// TIA Portal V16 export
// export: Created 2022-07-21T09:35:14.5212503Z, ExportSetting WithDefaults, DisplayName Totally Integrated Automation Portal, DisplayVersion V16 Update 4, DisplayName TIA Portal Version Control Interface, DisplayVersion V16 Update 2, DisplayName TIA Portal Openness, DisplayVersion V16 Update 4, DisplayName SINAMICS Startdrive Advanced, DisplayVersion V16 Update 5, DisplayName SINAMICS Startdrive G130, G150, S120, S150, SINAMICS MV, S210, DisplayVersion V16 Update 5, DisplayName SINAMICS Startdrive G110M, G120, G120C, G120D, G120P, G115D, DisplayVersion V16 Update 5, DisplayName STEP 7 Professional, DisplayVersion V16 Update 4, DisplayName STEP 7 Safety, DisplayVersion V16, DisplayName WinCC Advanced, DisplayVersion V16 Update 4
FUNCTION_BLOCK "LAxisBasics_AxisBasics_SyncAxis"   // FB833, FBD
TITLE = SyncAxis / Obsługa SyncAxis
{ S7_Optimized_Access := 'TRUE' }
AUTHOR : ArSc
FAMILY : LAxisBasics
VERSION : 1.1
// stored: AutoNumber false, IsIECCheckEnabled false, IsRetainMemResEnabled false, MemoryReserve 100, SetENOAutomatically false, UDAEnableTagReadback false
   VAR_INPUT
      axis : TO_SynchronousAxis;
      powerEnable : Bool;
      powerStartMode : DInt := 1;
      powerStopMode : Int := 0;
      resetExecute : Bool;
      resetRestart : Bool := false;
      homeExecute : Bool;
      homePosition : LReal;
      homeMode : Int;
      jogForward : Bool;
      jogBackward : Bool;
      jogVelocity : LReal := 100.0;   // [mm/s]
      jogAcceleration : LReal := -1.0;   // [mm/s²]
      jogDeceleration : LReal := -1.0;   // [mm/s²]
      jogJerk : LReal := -1.0;   // [mm/s³]
      jogPositionControlled : Bool := true;
   END_VAR
   VAR_OUTPUT
      powerStatus : Bool;
      powerBusy : Bool;
      resetDone : Bool;
      resetBusy : Bool;
      homeDone : Bool;
      homeBusy : Bool;
      jogInVelocity : Bool;
      jogBusy : Bool;
      commandAborted : Bool;
      error : Bool;
      errorID : Word;
      statusID : Int;
      axisData { ExternalAccessible := 'False'; ExternalVisible := 'False'; ExternalWritable := 'False'} : "LAxisBasics_typeAxisData";
   END_VAR
   VAR
      instMcPower { S7_SetPoint := 'True'} : MC_POWER;
      instMcReset { S7_SetPoint := 'True'} : MC_RESET;
      instMcHome { S7_SetPoint := 'True'} : MC_HOME;
      instMcMoveJog { S7_SetPoint := 'True'} : MC_MOVEJOG;
      statCommandAborted : Array[#ARRAY_BEGIN..#ARRAY_END] of Bool;
      statError : Array[#ARRAY_BEGIN..#ARRAY_END] of Bool;
      statErrorID : Array[#ARRAY_BEGIN..#ARRAY_END] of Word;
   END_VAR
   VAR_TEMP
      tempDwordCommandAborted : DWord;
      tempDwordError : DWord;
      tempCount : Int;
   END_VAR
   VAR CONSTANT
      ARRAY_BEGIN : Int := 1;
      ARRAY_END : Int := 32;
      ERROR_DEFAULT : Bool := false;
      ERRORID_DEFAULT : Word := 16#0;
      STATUSID_DEFAULT : Int := 0;
   END_VAR
BEGIN

REGION Network 1 (SCL): Information / Informacja
   //=============================================================================
   //SIEMENS AG
   //(c)Copyright 2016 All Rights Reserved
   //-----------------------------------------------------------------------------
   //Library:       Axis Basics
   //Tested with:   S7-1500T V2.5
   //Engineering:   TIA Portal V15
   //Restrictions:  Motion Control Library V4.0
   //Requirements:  S7-1500(T)
   //Functionality: Basic axis control and data collection of TO_SynchronousAxis
   //-----------------------------------------------------------------------------
   //Change log table:
   //Version  Date       Expert in charge Changes applied
   //01.01.00 17.04.2018 ArSc             -
   //01.00.00 26.07.2017 ArSc             First released version
   //=============================================================================
END_REGION

REGION Network 2: Power / Zasilanie
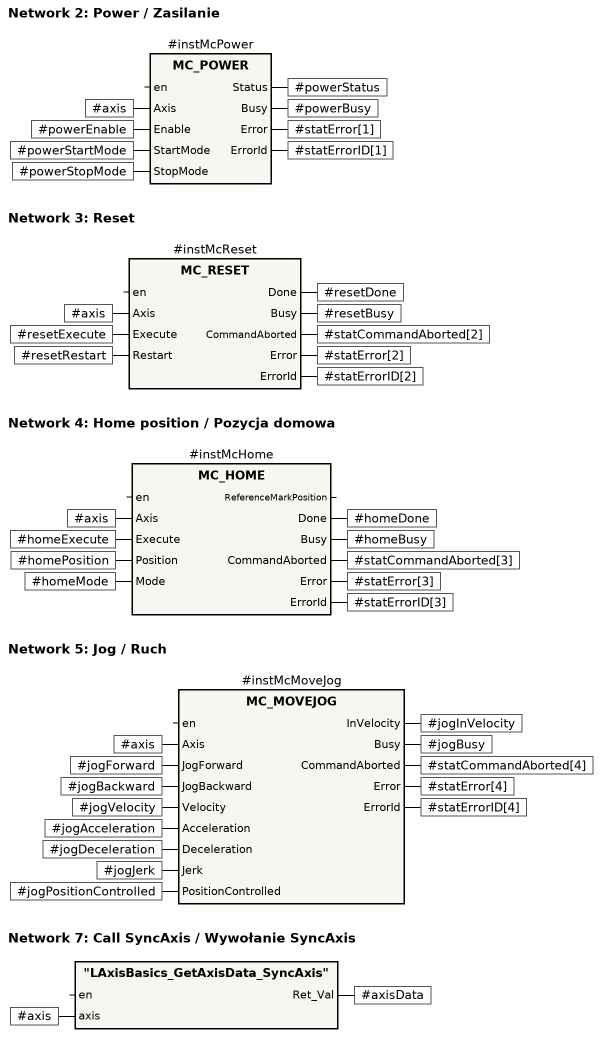
   #instMcPower(Axis := #axis,   // MC_POWER
                Enable := #powerEnable,
                StartMode := #powerStartMode,
                StopMode := #powerStopMode,
                Status => #powerStatus,
                Busy => #powerBusy,
                Error => #statError[1],
                ErrorId => #statErrorID[1]);
END_REGION

REGION Network 3: Reset
   #instMcReset(Axis := #axis,   // MC_RESET
                Execute := #resetExecute,
                Restart := #resetRestart,
                Done => #resetDone,
                Busy => #resetBusy,
                CommandAborted => #statCommandAborted[2],
                Error => #statError[2],
                ErrorId => #statErrorID[2]);
END_REGION

REGION Network 4: Home position / Pozycja domowa
   #instMcHome(Axis := #axis,   // MC_HOME
               Execute := #homeExecute,
               Position := #homePosition,
               Mode := #homeMode,
               Done => #homeDone,
               Busy => #homeBusy,
               CommandAborted => #statCommandAborted[3],
               Error => #statError[3],
               ErrorId => #statErrorID[3]);
END_REGION

REGION Network 5: Jog / Ruch
   #instMcMoveJog(Axis := #axis,   // MC_MOVEJOG
                  JogForward := #jogForward,
                  JogBackward := #jogBackward,
                  Velocity := #jogVelocity,
                  Acceleration := #jogAcceleration,
                  Deceleration := #jogDeceleration,
                  Jerk := #jogJerk,
                  PositionControlled := #jogPositionControlled,
                  InVelocity => #jogInVelocity,
                  Busy => #jogBusy,
                  CommandAborted => #statCommandAborted[4],
                  Error => #statError[4],
                  ErrorId => #statErrorID[4]);
END_REGION

REGION Network 6 (SCL): Outputs / Wyjścia
   //General output signals

   //Reset output signals
   #commandAborted := False;
   #error := False;
   #errorID := #ERRORID_DEFAULT;
   #statusID := #STATUSID_DEFAULT;

   //Transfer ARRAY to DWORD
   GATHER(IN:=#statCommandAborted,
          OUT=>#tempDwordCommandAborted);
   GATHER(IN:=#statError,
          OUT=>#tempDwordError);

   //Check for errors or command aborts
   IF (#tempDwordError > DWORD#0)
   THEN
     //Select error information
     FOR #tempCount := #ARRAY_BEGIN TO #ARRAY_END
     DO
       IF (#statError[#tempCount] = True)
       THEN
         #error := True;
         #errorID := #statErrorID[#tempCount];
         #statusID := #tempCount;
         EXIT;
       END_IF;
     END_FOR;
   ELSIF (#tempDwordCommandAborted > DWORD#0)
   THEN
     //Select command aborted information
     FOR #tempCount := #ARRAY_BEGIN TO #ARRAY_END
     DO
       IF (#statCommandAborted[#tempCount] = True)
       THEN
         #commandAborted := True;
         #errorID := #statErrorID[#tempCount];
         #statusID := #tempCount;
         EXIT;
       END_IF;
     END_FOR;
   END_IF;
END_REGION

REGION Network 7: Call SyncAxis / Wywołanie SyncAxis
   #axisData := "LAxisBasics_GetAxisData_SyncAxis"(axis := #axis);
END_REGION
END_FUNCTION_BLOCK
